Fanuc KAREL source: ko00072.KL

-- PROVISIONAL review KL for V770-1; original PC SHA256 87a385f5a491b27e5a36fa3bb036fffc2109ef331c685d5c9f0f819cd4d26af6
-- Incomplete behavior may be omitted. Consult companion uncertainty JSON. Do not deploy.
PROGRAM KO00072
%NOLOCKGROUP
BEGIN
  -- UNRESOLVED_PC offsets 5-12; opcodes 9D,23
  -- UNRESOLVED_PC offsets 17-66; opcodes 27,22,1C,27,49,7E,AD,22,31,7E,4A
  -- UNRESOLVED_PC offsets 71-75; opcodes 7F
END KO00072
